KUKA KRL data list: G1_Prog.dat

&ACCESS RVO
DEFDAT  G1_PROG
;FOLD EXTERNAL DECLARATIONS;%{PE}%MKUKATPBASIS,%CEXT,%VCOMMON,%P
;FOLD BASISTECH EXT;%{PE}%MKUKATPBASIS,%CEXT,%VEXT,%P
EXT  BAS (BAS_COMMAND  :IN,REAL  :IN )

DECL INT XTOOLBASE=3 ; ou o n?mero real da sua base
DECL INT XTOOL=3
DECL INT NextPos

DECL INT Z_Offset=50
DECL INT Angle_Offset=45

DECL POS RECOLHA={X -53.7200,Y -200.000,Z 133.000,C -90.0000}
DECL POS Matrix_Pos1={X 100.000,Y 200.000,Z 133.000,C 0.0}
DECL POS Matrix_Pos2={X 20.0000,Y 200.000,Z 133.000,C 0.0}
DECL POS Matrix_Pos3={X -60.0000,Y 200.000,Z 133.000,C 0.0}
DECL POS Matrix_Pos4={X 100.000,Y 120.000,Z 133.000,C 0.0}
DECL POS Matrix_Pos5={X 20.0000,Y 120.000,Z 133.000,C 0.0}
DECL POS Matrix_Pos6={X -60.0000,Y 120.000,Z 133.000,C 0.0}
DECL POS Matrix_Pos7={X 100.000,Y 40.0000,Z 133.000,C 0.0}
DECL POS Matrix_Pos8={X 20.0000,Y 40.0000,Z 133.000,C 0.0}
DECL POS Matrix_Pos9={X -60.0000,Y 40.0000,Z 133.000,C 0.0}


;ENDFOLD (BASISTECH EXT)
;FOLD USER EXT;%{E}%MKUKATPUSER,%CEXT,%VEXT,%P
;Make your modifications here

;ENDFOLD (USER EXT)
;ENDFOLD (EXTERNAL DECLARATIONS)
DECL MODULEPARAM_T LAST_TP_PARAMS={PARAMS[] "Kuka.PointName=Matrix_Pos1; Kuka.FrameData.base_no=2; Kuka.FrameData.tool_no=1; Kuka.FrameData.ipo_frame=#BASE; Kuka.isglobalpoint=False; Kuka.MoveDataName=CPDAT1; Kuka.MovementData.cb={AUX_PT {ORI #CONSIDER,E1 #CONSIDER,E2 #CONSIDER,E3 #CONSIDER,E4 #CONSIDER,E5 #CONSIDER,E6 #CONSIDER},TARGET_PT {ORI #INTERPOLATE,E1 #INTERPOLATE,E2 #INTERPOLATE,E3 #INTERPOLATE,E4 #INTERPOLATE,E5 #INTERPOLATE,E6 #INTERPOLATE}}; Kuka.MovementData.apo_fac=50; Kuka.MovementData.apo_dist=500; Kuka.MovementData.axis_acc=100; Kuka.MovementData.axis_vel=100; Kuka.MovementData.circ_typ=#BASE; Kuka.MovementData.jerk_fac=50; Kuka.MovementData.ori_typ=#VAR; Kuka.MovementData.vel=2; Kuka.MovementData.acc=100; Kuka.MovementData.exax_ign=0; Kuka.VelocityPath=2; Kuka.BlendingEnabled=True; Kuka.APXEnabled=False; Kuka.CurrentCDSetIndex=0; Kuka.VelocityFieldEnabled=False; Kuka.ColDetectFieldEnabled=False; Kuka.MovementParameterFieldEnabled=False; Kuka.IsAngleEnabled=False; Kuka.MoveDataPtpName=PDAT4; Kuka.MovementDataPdat.apo_mode=#CDIS; Kuka.MovementDataPdat.apo_dist=500; Kuka.VelocityPtp=100  "}
DECL PDAT PPDAT={VEL 100.000,ACC 100.000,APO_DIST 500.000,APO_MODE #CDIS,GEAR_JERK 100.000,EXAX_IGN 0}
DECL FDAT FBase={TOOL_NO 3,BASE_NO 3,IPO_FRAME #BASE,POINT2[] " "}

ENDDAT
